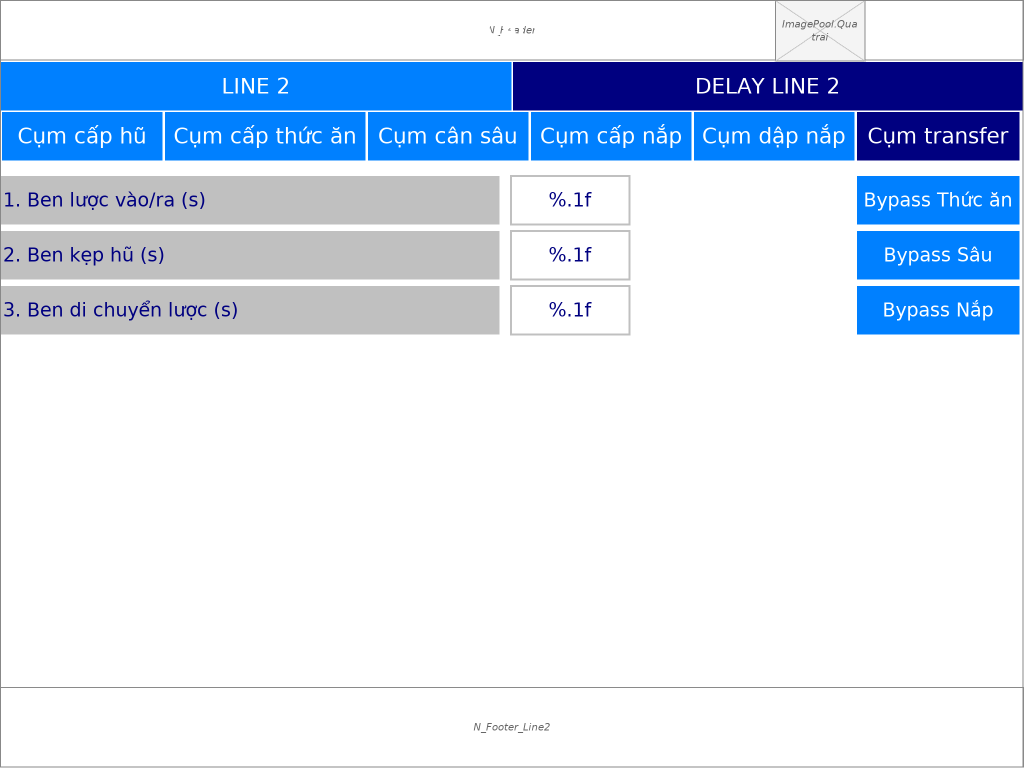
VISUALIZATION N_Setting_Delay_Tranfer2  // 1024x768
    Frame (0,687 1024x80)
        shows N_Footer_Line2()
    Frame (0,0 1024x60)
        shows N_Header()
    Textfield (353,4 420x50), "MÀN HÌNH CÀI KHOẢNG TRỄ LINE 2"
    Rectangle (0,175 500x50), "1. Ben lược vào/ra (s)"
    Rectangle (0,230 500x50), "2. Ben kẹp hũ (s)"
    Rectangle (0,285 500x50), "3. Ben di chuyển lược (s)"
    Group (0,61 1023x100)
        Rectangle (0,0 512x50), "LINE 2"
            OnMouseClick: change screen: N_Setting_Line2
        Rectangle (1,50 162x50), "Cụm cấp hũ"
            OnMouseClick: change screen: N_Setting_Delay_JarSupply2
        Rectangle (164,50 202x50), "Cụm cấp thức ăn"
            OnMouseClick: change screen: N_Setting_Delay_FoodSupply2
        Rectangle (367,50 162x50), "Cụm cân sâu"
            OnMouseClick: change screen: N_Setting_Delay_WorwWeight2
        Rectangle (530,50 162x50), "Cụm cấp nắp"
            OnMouseClick: change screen: N_Setting_Delay_LidSupply2
        Rectangle (693,50 162x50), "Cụm dập nắp"
            OnMouseClick: change screen: N_Setting_Delay_LidPressing2
        Rectangle (856,50 164x50), "Cụm transfer"
            OnMouseClick: change screen: N_Setting_Delay_Tranfer2
        Rectangle (512,0 511x50), "DELAY LINE 2"
            OnMouseClick: change screen: N_Setting_Delay_JarSupply2
    Image (775,0 90x61), image: ImagePool.Qua trai
        OnMouseClick: change screen: N_Setting_Delay_Tranfer1
    Rectangle (510,175 120x50), "%.1f", text variable: PR_Line02.fTimer_Comb
        OnMouseClick: write PR_Line02.fTimer_Comb via VisuDialogs.Numpad
    Rectangle (510,230 120x50), "%.1f", text variable: PR_Line02.fTimer_Clip
        OnMouseClick: write PR_Line02.fTimer_Clip via VisuDialogs.Numpad
    Rectangle (510,285 120x50), "%.1f", text variable: PR_Line02.fTimer_Move_Comb
        OnMouseClick: write PR_Line02.fTimer_Move_Comb via VisuDialogs.Numpad
    Rectangle (856,175 164x50), "Bypass Thức ăn"
        toggle PR_Line02.bypassFood
    Rectangle (856,230 164x50), "Bypass Sâu"
        toggle PR_Line02.bypassWorm
    Rectangle (856,285 164x50), "Bypass Nắp"
        toggle PR_Line02.bypassLid
END_VISUALIZATION

(* stored: Version 1.1.0.1, ProductVersion 3.1.4024.12
   Visu N_Setting_Delay_Tranfer2: Id {dbec6ffe-4ac5-475b-8abb-60287a4f509e} *)
